Fanuc KAREL source: kb00145.KL

PROGRAM KB00145
%STACKSIZE=65535
%PRIORITY=65535
%NOLOCKGROUP
VAR
P1 : STRING[80]
P2 : STRING[80]
P3 : INTEGER
BEGIN
P1='A'
P2='A'
P3=1
REMOVE_DICT(P1,P2,P3)
END KB00145
